DATA_BLOCK "bioPoT.DB"
{ S7_Optimized_Access := 'TRUE' }
VERSION : 1.0
// Batch I/O Polygon Table Data Block:
// by Woermann Automation
NON_RETAIN
   VAR RETAIN
      PoT : Array[0..15] of "bioPoT.DT";
   END_VAR

BEGIN

END_DATA_BLOCK

